{attribute 'linkalways'} 
{attribute 'no_explicit_call' := 'This FB is a CLASS and must be accessed using methods or properties'}
{attribute 'enable_dynamic_creation'}
FUNCTION_BLOCK ABSTRACT UserDefinedDatatypeBase EXTENDS DatatypeBase IMPLEMENTS I_UserDefinedDatatype
VAR
END_VAR

PROPERTY PUBLIC ABSTRACT Identifier : T_MAXSTRING
GET
END_GET
END_PROPERTY

METHOD PUBLIC IsEquivalentTo : BOOL
VAR_INPUT
	Datatype : I_Datatype;
END_VAR
VAR
	datatypeAsUdt : I_UserDefinedDatatype;
END_VAR
IF NOT Datatype.Root.TryResolveAsUserDefinedDatatype(datatypeAsUdt) THEN
	RETURN;
END_IF

IF datatypeAsUdt.Identifier <> Identifier THEN
	RETURN;
END_IF

IsEquivalentTo := SUPER^.IsEquivalentTo(Datatype);
END_METHOD

PROPERTY PUBLIC IsUserDefined : BOOL
GET
IsUserDefined := TRUE;
END_GET
END_PROPERTY

METHOD PROTECTED OnSerializeTypeWith
VAR_INPUT
	Serializer : I_Serializer;
END_VAR
SUPER^.OnSerializeTypeWith(Serializer);
Serializer.AddKeyString('identifier',Identifier);
END_METHOD

METHOD PUBLIC TryCopyFrom : BOOL
VAR_INPUT
	Source : I_Datatype;
END_VAR
VAR
	sourceAsUdt : I_UserDefinedDatatype;
END_VAR
IF NOT __QUERYINTERFACE(Source, sourceAsUdt) THEN
	RETURN;
END_IF

IF sourceAsUdt.Identifier <> Identifier THEN
	RETURN;
END_IF

TryCopyFrom := SUPER^.TryCopyFrom(Source);
END_METHOD

METHOD PUBLIC TryResolveAsUserDefinedDatatype : BOOL
VAR_INPUT
	Destination : REFERENCE TO I_UserDefinedDatatype;
END_VAR
Destination := THIS^;
TryResolveAsUserDefinedDatatype := TRUE;
END_METHOD

END_FUNCTION_BLOCK

(* stored: Version 1.1.0.1, ProductVersion 3.1.4026.18
   POU UserDefinedDatatypeBase: Id {fd645b0d-4a81-0ada-1363-d0e819ed505d}, SpecialFunc None
   Folder Protected: Id {82160199-9ad7-0918-0742-b6cf882ff325}
   Property Identifier: Id {f8ae4709-f25c-0671-045d-981221625415}
   Get Get: Id {d35650fc-dbe8-0a9d-0fef-f637b653bb56}
   Method IsEquivalentTo: Id {c436fbfa-5783-0250-1ee0-e968f743b1ab}
   Property IsUserDefined: Id {bec904ee-ddc4-4330-9cbc-67c183e16939}
   Get Get: Id {6d8d4eb1-bb1d-412d-8e85-9da1c88e349f}
   Method OnSerializeTypeWith: Id {efeaa587-6602-09b9-2f80-a5828c650546}
   Method TryCopyFrom: Id {acc31a0e-04bd-4623-9e71-5f78de76eab3}
   Method TryResolveAsUserDefinedDatatype: Id {17304df6-1666-0527-3373-79f0c5b364f7} *)
